Staubli VAL3: ENTRYBOX.pjx

--- ENTRYBOX.pjx ---
Parameters version=s7.1 stackSize=5000 millimeterUnit=true
Program file=_findBorders.pgx
Program file=_GetUserInput.pgx
Program file=_handleCounter.pgx
Program file=_removeChar.pgx
Program file=_resizeData.pgx
Program file=_writeTxtBoxVal.pgx
Program file=create.pgx
Program file=display.pgx
Program file=eraseField.pgx
Program file=getCaption.pgx
Program file=getErrorMessage.pgx
Program file=getFieldValue.pgx
Program file=handle.pgx
Program file=handleBtype.pgx
Program file=handleLtype.pgx
Program file=handleNtype.pgx
Program file=setFieldValue.pgx
Program file=setListOfItems.pgx
Program file=start.pgx
Program file=stop.pgx
Data file=EntryBox.dtx
Library alias=pw path=Disk://Tracking/Templates/GenericPage/GenericPage.pjx
Library alias=up path=Disk://Tracking/Tools/userPage/userPage.pjx
Library alias=ut path=Disk://Tracking/Tools/util/util.pjx

--- ENTRYBOX.dtx ---
num nDummy
num nFocused
num nLblPosX[3]
  [1] = 22
num nLblPosY[3] = 6
public num nNumOfLabel = 3
public num nNumOfTxtBox = 10
num nPageUpCol
num nPageUpRow
num nTxtFocused
num nTxtMaxVal[10]
  [0] = 1000
  [1] = 1000
  [2] = 200
  [4] = 200
  [5] = 20
  [6] = 99
  [8] = 999
  [9] = 999
num nTxtMinVal[10]
  [0] = -1000
  [1] = -1000
  [2] = 5
  [4] = 1
  [5] = 1
  [6] = 1
num nTxtPosX[10]
  [6] = 22
  [7] = 22
  [8] = 22
  [9] = 22
num nTxtPosY[10]
  [0] = 1
  [1] = 2
  [2] = 3
  [3] = 4
  [4] = 7
  [5] = 8
  [6] = 1
  [7] = 3
  [8] = 4
  [9] = 5
num nVIDEOCUSTOM = 2
num nVIDEOINVERSED = 1
num nVIDEONORMAL
string sErrMsgList[6]
  [1] = "The library *\../* couldn't not be loaded because of the error code n°*"
  [2] = "Error from definition library *\../*."
  [3] = "The variable sListItem* of the definition library is not defined."
  [4] = "The  caption '*\../*'  does not exist"
string sErrorMessage = "The library GenericWin couldn't not be loaded because of the error code n°30"
string sListItems
bool bDrawFrame
public mdesc mNomSpeed = {blend=off}

--- getFieldValue.pgx ---
public program getFieldValue(string x_sCaption, string& x_sValue[], num x_nError)
  local num l_i
  local bool l_bFound
  local bool l_bQuit
begin
  // This program returns the value of the field passed as parameter
  //
  // Input Param
  //  x_sCaption      : Name of the field
  //
  // Output Param
  //  x_sValue      : Current value
  //  x_nError      : Error code
  //                = 0 success
  //                = 1 Caption  not found
  //Created 21/12/05                              CCUR
  //--------------------------------------------------------------
  x_nError=0
  // Search if label passed as parameter is known
  l_i=0
  do
    l_bFound=(x_sCaption==pw:sTxtBoxCaption[l_i])
    l_i=l_i+1
  until (l_bFound or (l_i>=nNumOfTxtBox))
  //
  if l_bFound
    x_sValue=pw:sTxtBoxVal[l_i-1]
  else
    x_nError=4
    // Prepare clear text error message
    call ut:addStrToString(sErrMsgList[x_nError],sErrorMessage,"",x_sCaption)
  endIf
end
